FUNCTION_BLOCK FB_Timer IMPLEMENTS I_Timer
VAR
	_Timer: TON;

	_done: BOOL;
	_busy: BOOL;
	_free: BOOL := TRUE;
END_VAR

PROPERTY PUBLIC Busy : BOOL
GET
Busy := _busy;
END_GET
END_PROPERTY

PROPERTY PUBLIC Done : BOOL
GET
Done := _done;
END_GET
END_PROPERTY

PROPERTY PUBLIC ElapsedTime : TIME
GET
ElapsedTime := _Timer.ET;
END_GET
END_PROPERTY

METHOD Execute
_Timer();

IF _Timer.Q THEN
	_done := TRUE;
	_busy := FALSE;
END_IF
END_METHOD

METHOD Register : BOOL
Register := TIMERS.Manager.Register(THIS^);
END_METHOD

METHOD PUBLIC Reset
_Timer(IN := FALSE);

_done := FALSE;
_busy := FALSE;
_free := TRUE;
END_METHOD

METHOD PUBLIC Start
VAR_INPUT
	delay: TIME;
END_VAR
IF _free THEN
	_Timer(IN := FALSE);
	_Timer(IN := TRUE,
			PT := delay);

	_busy := TRUE;
	_done := FALSE;
	_free := FALSE;
END_IF
END_METHOD

END_FUNCTION_BLOCK

(* stored: Version 1.1.0.1, ProductVersion 3.1.4024.9
   POU FB_Timer: Id {cf83e778-4f9b-49e1-ad4e-e52c03835e4c}, SpecialFunc None
   Property Busy: Id {c9fb5124-bc69-4b54-b1d3-13ba468da833}
   Get Get: Id {afb43b8c-9eeb-4907-9e48-28ecc2779509}
   Property Done: Id {886cc76c-76a9-404e-bdff-86b318cdb24d}
   Get Get: Id {56338a4a-6803-4dde-990f-fb086704f76d}
   Property ElapsedTime: Id {e7749abd-8541-461b-b5f3-0649c7956556}
   Get Get: Id {8cf9ecfd-0ba2-4642-96c9-61d2e12f2716}
   Method Execute: Id {54c9b7de-94dc-4c2c-8a06-10b15fab4bcd}
   Method Register: Id {06a570ed-0461-4998-a0bf-22c2f135ba1f}
   Method Reset: Id {fb1af245-de7f-4d60-be89-f5091a8e41b6}
   Method Start: Id {3720fc15-1a4e-4e99-8c08-e8707e20b76a} *)
